% RSLogix 500 project I2P JOB 23 - ALEXANDER_LOYND_BAK120.RSS, saved by version 10.00.00.00 %
PROJECT "ML06A"    % processor: Bul.1763 MicroLogix 1100 Series B %

PROGRAM FILES
  LAD 2   18 rungs

DATA FILES
  O0 OUTPUT  4 elements
  I1 INPUT  6 elements
  S2 STATUS  66 elements
  B3 BINARY  1 elements
  T4 TIMER  1 elements
  C5 COUNTER  2 elements
  R6 CONTROL  1 elements
  N7 INTEGER  1 elements
  F8 FLOAT  1 elements

LADDER 2
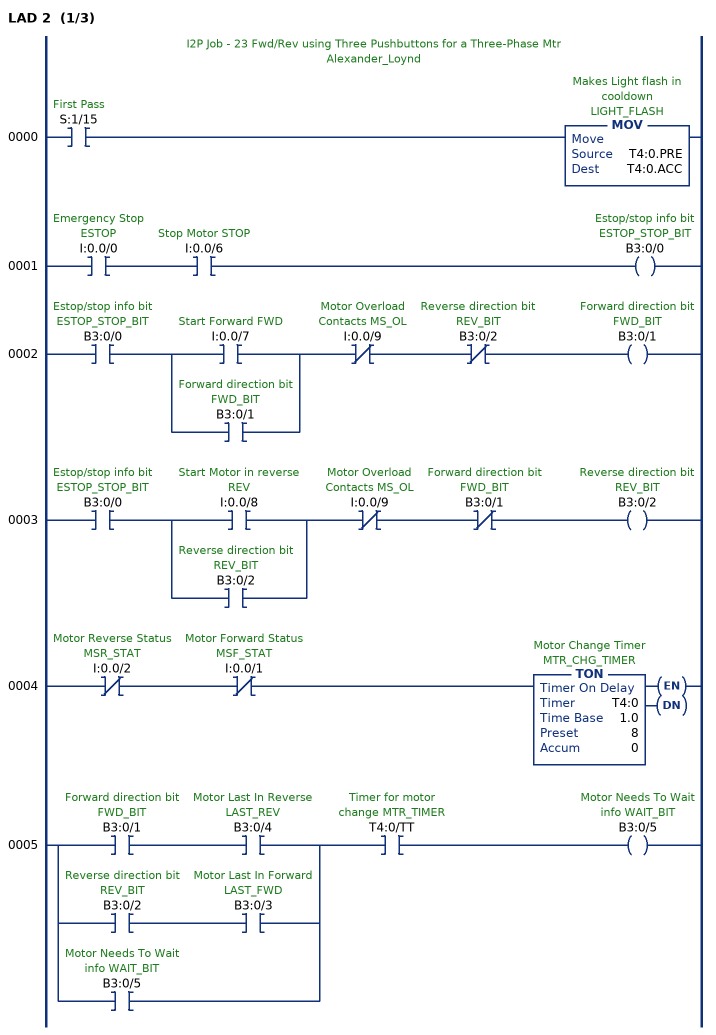
% Rung: 0 %
% I2P Job - 23 Fwd/Rev using Three Pushbuttons for a Three-Phase Mtr
% Alexander_Loynd %
SOR XIC S:1/15 MOV T4:0.PRE T4:0.ACC EOR
%   S:1/15  "First Pass" %
%   T4:0  MTR_CHG_TIMER  "Motor Change Timer" %
%   T4:0.ACC  LIGHT_FLASH  "Makes Light flash in cooldown" %
% Rung: 1 %
SOR XIC I:0.0/0 XIC I:0.0/6 OTE B3:0/0 EOR
%   I:0.0/0  ESTOP  "Emergency Stop" %
%   I:0.0/6  STOP  "Stop Motor" %
%   B3:0/0  ESTOP_STOP_BIT  "Estop/stop info bit" %
% Rung: 2 %
SOR XIC B3:0/0 BST XIC I:0.0/7 NXB XIC B3:0/1 BND XIO I:0.0/9 XIO B3:0/2 OTE B3:0/1 EOR
%   B3:0/0  ESTOP_STOP_BIT  "Estop/stop info bit" %
%   I:0.0/7  FWD  "Start Forward" %
%   B3:0/1  FWD_BIT  "Forward direction bit" %
%   I:0.0/9  MS_OL  "Motor Overload Contacts" %
%   B3:0/2  REV_BIT  "Reverse direction bit" %
% Rung: 3 %
SOR XIC B3:0/0 BST XIC I:0.0/8 NXB XIC B3:0/2 BND XIO I:0.0/9 XIO B3:0/1 OTE B3:0/2 EOR
%   B3:0/0  ESTOP_STOP_BIT  "Estop/stop info bit" %
%   I:0.0/8  REV  "Start Motor in reverse" %
%   B3:0/2  REV_BIT  "Reverse direction bit" %
%   I:0.0/9  MS_OL  "Motor Overload Contacts" %
%   B3:0/1  FWD_BIT  "Forward direction bit" %
% Rung: 4 %
SOR XIO I:0.0/2 XIO I:0.0/1 TON T4:0 1.0 8 0 EOR
%   I:0.0/2  MSR_STAT  "Motor Reverse Status" %
%   I:0.0/1  MSF_STAT  "Motor Forward Status" %
%   T4:0  MTR_CHG_TIMER  "Motor Change Timer" %
% Rung: 5 %
SOR BST XIC B3:0/1 XIC B3:0/4 NXB BST XIC B3:0/2 XIC B3:0/3 NXB XIC B3:0/5 BND BND XIC T4:0/TT OTE B3:0/5 EOR
%   B3:0/1  FWD_BIT  "Forward direction bit" %
%   B3:0/4  LAST_REV  "Motor Last In Reverse" %
%   B3:0/2  REV_BIT  "Reverse direction bit" %
%   B3:0/3  LAST_FWD  "Motor Last In Forward" %
%   B3:0/5  WAIT_BIT  "Motor Needs To Wait info" %
%   T4:0/TT  MTR_TIMER  "Timer for motor change" %

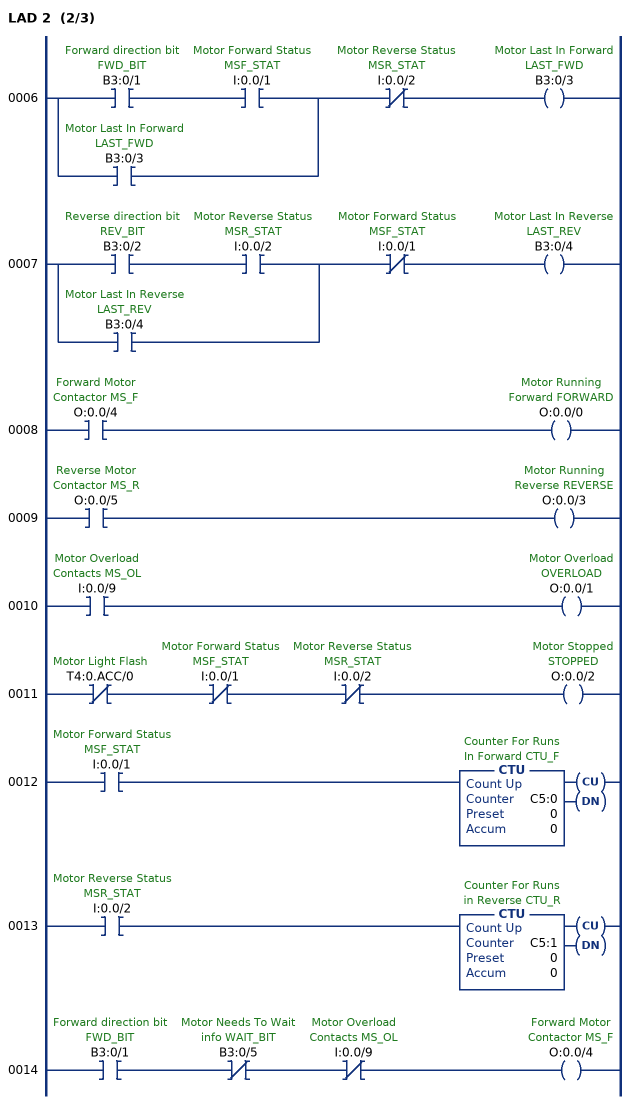
% Rung: 6 %
SOR BST XIC B3:0/1 XIC I:0.0/1 NXB XIC B3:0/3 BND XIO I:0.0/2 OTE B3:0/3 EOR
%   B3:0/1  FWD_BIT  "Forward direction bit" %
%   I:0.0/1  MSF_STAT  "Motor Forward Status" %
%   B3:0/3  LAST_FWD  "Motor Last In Forward" %
%   I:0.0/2  MSR_STAT  "Motor Reverse Status" %
% Rung: 7 %
SOR BST XIC B3:0/2 XIC I:0.0/2 NXB XIC B3:0/4 BND XIO I:0.0/1 OTE B3:0/4 EOR
%   B3:0/2  REV_BIT  "Reverse direction bit" %
%   I:0.0/2  MSR_STAT  "Motor Reverse Status" %
%   B3:0/4  LAST_REV  "Motor Last In Reverse" %
%   I:0.0/1  MSF_STAT  "Motor Forward Status" %
% Rung: 8 %
SOR XIC O:0.0/4 OTE O:0.0/0 EOR
%   O:0.0/4  MS_F  "Forward Motor Contactor" %
%   O:0.0/0  FORWARD  "Motor Running Forward" %
% Rung: 9 %
SOR XIC O:0.0/5 OTE O:0.0/3 EOR
%   O:0.0/5  MS_R  "Reverse Motor Contactor" %
%   O:0.0/3  REVERSE  "Motor Running Reverse" %
% Rung: 10 %
SOR XIC I:0.0/9 OTE O:0.0/1 EOR
%   I:0.0/9  MS_OL  "Motor Overload Contacts" %
%   O:0.0/1  OVERLOAD  "Motor Overload" %
% Rung: 11 %
SOR XIO T4:0.ACC/0 XIO I:0.0/1 XIO I:0.0/2 OTE O:0.0/2 EOR
%   T4:0.ACC/0  "Motor Light Flash" %
%   I:0.0/1  MSF_STAT  "Motor Forward Status" %
%   I:0.0/2  MSR_STAT  "Motor Reverse Status" %
%   O:0.0/2  STOPPED  "Motor Stopped" %
% Rung: 12 %
SOR XIC I:0.0/1 CTU C5:0 0 0 EOR
%   I:0.0/1  MSF_STAT  "Motor Forward Status" %
%   C5:0  CTU_F  "Counter For Runs In Forward" %
% Rung: 13 %
SOR XIC I:0.0/2 CTU C5:1 0 0 EOR
%   I:0.0/2  MSR_STAT  "Motor Reverse Status" %
%   C5:1  CTU_R  "Counter For Runs in Reverse" %
% Rung: 14 %
SOR XIC B3:0/1 XIO B3:0/5 XIO I:0.0/9 OTE O:0.0/4 EOR
%   B3:0/1  FWD_BIT  "Forward direction bit" %
%   B3:0/5  WAIT_BIT  "Motor Needs To Wait info" %
%   I:0.0/9  MS_OL  "Motor Overload Contacts" %
%   O:0.0/4  MS_F  "Forward Motor Contactor" %

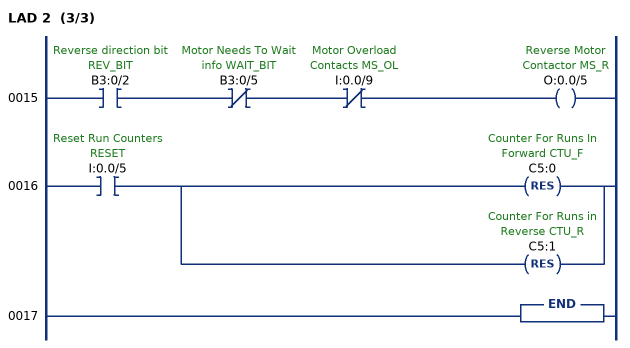
% Rung: 15 %
SOR XIC B3:0/2 XIO B3:0/5 XIO I:0.0/9 OTE O:0.0/5 EOR
%   B3:0/2  REV_BIT  "Reverse direction bit" %
%   B3:0/5  WAIT_BIT  "Motor Needs To Wait info" %
%   I:0.0/9  MS_OL  "Motor Overload Contacts" %
%   O:0.0/5  MS_R  "Reverse Motor Contactor" %
% Rung: 16 %
SOR XIC I:0.0/5 BST RES C5:0 NXB RES C5:1 BND EOR
%   I:0.0/5  RESET  "Reset Run Counters" %
%   C5:0  CTU_F  "Counter For Runs In Forward" %
%   C5:1  CTU_R  "Counter For Runs in Reverse" %
% Rung: 17 %
SOR END EOR

OTHER DOCUMENTED ADDRESSES
  I:0.0/3  MODE_ON  "On Setting 3PSS"
  I:0.0/4  MODE_AUTO  "AUTO Setting 3PSS"
  MOV  
  PB1  "Start Motor"
  T4:0/DN  T4

DATA TABLE (non-zero values as saved)
DATA T4
% .PRE .ACC %
% T4:0 % 8 0
